FUNCTION_BLOCK PLCopenRemote IMPLEMENTS IPLCopenCallRemote, IPLCopenCallStatus
VAR_INPUT
  command : IPLCopenCommand;
END_VAR
VAR
  _PLCopenCallInternal : PLCopenRemoteInternal;
  status : IPLCopenCallStatus;
  _delegate : IPLCopenCallRemote;
  _nullRemote : PLCopenNullRemote;
END_VAR

PROPERTY Abort : BOOL
GET
abort := _PLCopenCallInternal.abort;
END_GET
SET
_PLCopenCallInternal.abort := abort;
END_SET
END_PROPERTY

PROPERTY Delegate : IPLCopenCallRemote
GET
IF _delegate <> 0 THEN
	Delegate := _delegate;
ELSE
	Delegate := _nullRemote;
END_IF
END_GET
SET
_delegate := Delegate;
END_SET
END_PROPERTY

{attribute 'monitoring' := 'call'}
PROPERTY RemoteStatus : PLCopenStatusBase
GET
RemoteStatus := _PLCopenCallInternal.status;
END_GET
SET
_PLCopenCallInternal.status := RemoteStatus;
END_SET
END_PROPERTY


METHOD ReportAborted : BOOL

// Copyright (c) 2024 Loupe (https://loupe.team), provided under the MIT License.

_PLCopenCallInternal.abort := TRUE;
Delegate.ReportAborted();
END_METHOD


METHOD ReportErrored : BOOL
VAR_INPUT
  ID : INT;
END_VAR

// Copyright (c) 2024 Loupe (https://loupe.team), provided under the MIT License.

CASE ID OF
  //Any of these statuses are invalid to return as an error.
  //Override to error
  	PLCopenStatusBase.BUSY,
	PLCopenStatusBase.ENABLED_WAITING,
	PLCopenStatusBase.ERR_OK:
    _PLCopenCallInternal.status := PLCopenStatusBase.ERROR;
ELSE
  //Any other status can be passed through
  _PLCopenCallInternal.status := ID;
END_CASE

IF delegate <> 0 THEN
	delegate.ReportErrored(_PLCopenCallInternal.status);
END_IF
END_METHOD


METHOD ReportFinished : BOOL

// Copyright (c) 2024 Loupe (https://loupe.team), provided under the MIT License.

_PLCopenCallInternal.status := PLCopenStatusBase.ERR_OK;

IF delegate <> 0 THEN
	delegate.ReportFinished();
END_IF
END_METHOD


METHOD Start : BOOL
VAR_INPUT
  Command : IPLCopenCommand;
END_VAR
 _PLCopenCallInternal.status := PLCopenStatusBase.ENABLED_WAITING;
command.RemoteExecute(THIS^);
END_METHOD

END_FUNCTION_BLOCK

(* stored: Version 1.1.0.1
   POU PLCopenRemote: Id {603500fb-9066-4ec5-b073-ea0871d605ca}, SpecialFunc None
   Property Abort: Id {c7641c67-ae0d-4596-b708-3691eb9c1d20}
   Get Get: Id {59c0b979-29c2-4ad1-b323-896aa956b7b1}
   Set Set: Id {3bc2a4d4-a0df-4a5d-87f3-0a319ab86ebb}
   Property Delegate: Id {bce0543c-2a05-0c7a-3389-99dd8eec4ed4}
   Get Get: Id {06008cca-71d3-05a3-20b6-395d0133b4b2}
   Set Set: Id {b5e3a340-0eb0-04ac-1f26-d0ac42dcb271}
   Property RemoteStatus: Id {27ee096e-7abf-4323-b731-6523795b731f}
   Get Get: Id {e2b3ab12-0ad9-4b99-adc0-fc57a956ef6f}
   Set Set: Id {1a539f5d-b4b2-467b-8226-4bf0c3488566}
   Method ReportAborted: Id {cbecde3e-63d7-41c9-90ae-249e6fdbfbdc}
   Method ReportErrored: Id {c6822c79-4afc-4bd0-8933-2b53beb26986}
   Method ReportFinished: Id {cf5564a2-2dcb-446f-9ce1-2b34ce737728}
   Method Start: Id {4e7a139b-9cbd-4971-b8b3-78113352ebfb} *)
